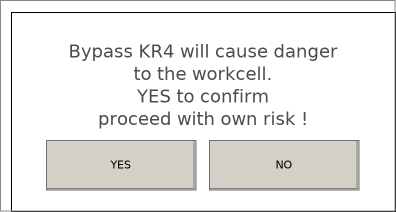
VISUALIZATION MSG_KR5_BP  // 396x212
    RoundedRectangle (11,12 385x200)
    Button (46,140 150x50), "YES"
        OnMouseClick: CloseDialog Dialog=MSG_KR5_BP, Result=No, NumpadKeypadSet=True
        OnMouseClick: execute { GVL.KR5_bypass := TRUE; }
    Button (209,140 150x50), "NO"
        OnMouseClick: execute { GVL.KR5_bypass := FALSE; }
        OnMouseClick: CloseDialog Dialog=MSG_KR5_BP, Result=No, NumpadKeypadSet=True
    Label (55,30 296x110), "Bypass KR4 will cause danger to the workcell. YES to confirm proceed with own risk !"
END_VISUALIZATION

(* stored: Version 1.1.0.1, ProductVersion 3.1.4024.12
   Visu MSG_KR5_BP: Id {89c2300c-29e4-48f0-8da1-57edd31b7e4b} *)
